// TIA Portal project "motor test code" (V20)

(* hardware
DEVICE "S7-1200 station_1"  S7-1200 Station
   slot 0: "Rack_0"  S7-1200 Rack  Rack  V1.0
   slot 1: "PLC_1"  CPU 1214C DC/DC/DC  6ES7 214-1AG40-0XB0  V4.6
   slot 2: "DI 8x24VDC/DQ 8xRelay_1"  SM 1223 DI8/DQ8 x relay  6ES7 223-1PH32-0XB0  V2.0
   slot 3: "AI 4x13BIT/AQ 2x14BIT_1"  SM 1234 AI4/AQ2  6ES7 234-4HE32-0XB0  V2.1
DEVICE "HMI_1"  KTP700 Basic PN
   slot 0: "HMI_1"  KTP700 Basic PN  6AV2 123-2GB03-0AX0  17.0.0.0
   slot 1: "HMI_RT_1"  KTP700 Basic PN  6AV2 123-2GB03-0AX0  17.0.0.0
   slot 5: "HMI_1.IE_CP_1"  PROFINET Interface  17.0.0.0
      slot 1: "PROFINET Interface_1"  PROFINET Interface
         slot 1: "Port_1"  Port
DEVICE "SINAMICS S_2"  SINAMICS S210
   slot 0: "Drive unit_2"  S210 PN  6SL3210-5HB10-4xFx  V5.2
      slot 1: "PROFINET interface"  PROFINET
      slot 3: "Ethernet commissioning interface"  LAN
   slot 0: "Drive control"  S210 PN
      slot 200: "Power Module_1"  Drive control  6SL3210-5HB10-4xFx
      slot 300: "Encoder evaluation_1"  Drive control  1FK2103-4AG0x-xMxx
      slot 400: "Measuring system_1"  Drive control  1FK2103-4AG0x-xMxx
      slot 1000: "Motor_1"  Drive control  1FK2103-4AG0x-xMxx
*)

// ===== PLC "PLC_1"  CPU 1214C DC/DC/DC =====

VAR_GLOBAL   // PLC tag table "Default tag table"
   "Brugaansturing_axis_IN" AT %I256.0 : "PD_TEL3_IN";
   "Brugaansturing_axis_OUT" AT %Q256.0 : "PD_TEL3_OUT";
   "ProgramCounter" AT %MW100 : Int;
   "em_stop" AT %I0.0 : Bool;
   "Reset Button" AT %I0.1 : Bool;
   "Homing sensor" AT %I0.2 : Bool;
   "Gate Closed" AT %I0.3 : Bool;
   "Gate Open" AT %I0.4 : Bool;
   "LightSwitch Front" AT %I0.5 : Bool;
   "LightSwitch Middle" AT %I0.6 : Bool;
   "Start Button" AT %I0.7 : Bool;
   "Stop Button" AT %I1.0 : Bool;
   "Open Gate" AT %Q0.0 : Bool;
   "Road_Yellow" AT %Q0.1 : Bool;
   "Road_Green" AT %Q0.2 : Bool;
   "Road_Red" AT %Q0.3 : Bool;
   "Noodstop Rood" AT %Q0.4 : Bool;
   "Noodstop Groen" AT %Q0.5 : Bool;
   "Autohome" AT %M1.1 : Bool;
   "JogForward" AT %M1.2 : Bool;
   "JogBackward" AT %M1.3 : Bool;
END_VAR

DATA_BLOCK "BrugAansturing_axis"   // DB1, Motion_DB
{ S7_Optimized_Access := 'TRUE' }
AUTHOR : SIMATIC
FAMILY : BasicMC
NAME : TO_PosAx
VERSION : 6.0
// stored: InstanceOfName TO_PositioningAxis
"TO_PositioningAxis"
BEGIN
   // Axis.Encoder.TelegramAddressOutCU = %Q256.0
   // Axis.Encoder.TelegramAddressInCU = %I256.0
   // Axis.Encoder.DoNameCU = Drive unit_2.Drive_control_Standard_telegram_3
   // Axis.Drive.TelegramAddressOutCU = %Q256.0
   // Axis.Drive.TelegramAddressInCU = %I256.0
   // Axis.Drive.TelegramType = 2
   // Axis.Drive.DoNameCU = Drive unit_2.Drive_control_Standard_telegram_3
   // Axis.Encoder.SelectedHscIndexCU = -1
   // Axis.LengthUnit.LastDistance = 1005
   // Axis.LengthUnitNormalized.Time = 1
   // Axis.LengthUnitNormalized.Distance = -2
   // Axis.Encoder.DbTypeCU = Classic
   // Axis.Drive.DbTypeCU = Classic
END_DATA_BLOCK

FUNCTION "Block_1" : Void   // FC1, SCL
{ S7_Optimized_Access := 'TRUE' }
VERSION : 0.1
BEGIN
   "MC_Home_DB"(Axis:="BrugAansturing_axis",
                Execute:="Autohome",
                Mode:=3);
   IF "BrugAansturing_axis".StatusBits.HomingDone THEN
       "Autohome" := 0
       ;
   END_IF;
END_FUNCTION

FUNCTION "my_function1" : Void   // FC2, SCL
{ S7_Optimized_Access := 'TRUE' }
VERSION : 0.1
BEGIN
   IF "JogForward"=TRUE THEN
       "MC_Halt_DB"(Axis := "BrugAansturing_axis",
                    Execute := FALSE);
       "MC_MoveVelocity_DB"(Axis := "BrugAansturing_axis",
                            Execute := TRUE,
                            Velocity := 40,
                            Direction := 0);

   ELSIF "JogBackward"=TRUE THEN
       "MC_Halt_DB"(Axis := "BrugAansturing_axis",
                    Execute := FALSE);
       "MC_MoveVelocity_DB"(Axis:="BrugAansturing_axis",
                              Execute:=TRUE,
                              Velocity:=-40,
                              Direction:=0);
     ELSE
         ;
         "MC_MoveVelocity_DB"(Axis := "BrugAansturing_axis",
                              Execute := FALSE);
         "MC_Halt_DB"(Axis:="BrugAansturing_axis",
                      Execute:=TRUE);

   END_IF;
END_FUNCTION

ORGANIZATION_BLOCK "Main"   // OB1, LAD, ProgramCycle
TITLE = "Main Program Sweep (Cycle)"
{ S7_Optimized_Access := 'TRUE' }
VERSION : 0.1
   VAR_INPUT
      Initial_Call : Bool;   // Initial call of this OB
      Remanence : Bool;   // =True, if remanent data are available
   END_VAR
BEGIN

REGION Network 1
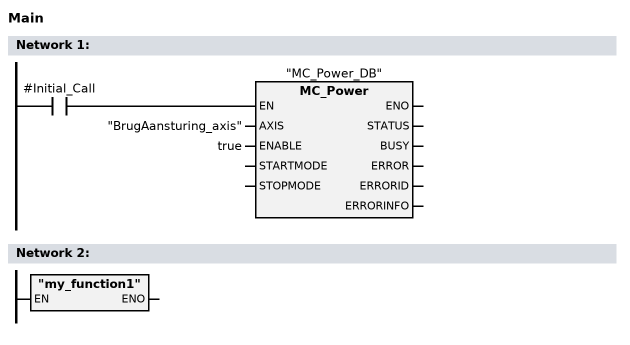
   IF #Initial_Call THEN
       "MC_Power_DB"(Axis := "BrugAansturing_axis", Enable := true);   // MC_Power
   END_IF;
END_REGION

REGION Network 2
   RUNG wire#powerrail
      "my_function1"()
   END_RUNG
   // the same network as SCL:
   "my_function1"();
END_REGION
END_ORGANIZATION_BLOCK

(* ===== HMI "HMI_RT_1" =====
system functions are stored by id; their names below are inferred from use
connection "HMI_Connection_1": ETHERNET, SMART_S7_1200_OMS

HMI tags "Default tag table"
   "HMI_Home" : UInt, internal
   "HMI_Debug" : UInt, internal
   "HMI_Manual overide" : UInt, internal
   "HMI_Nominal mode" : UInt, internal
   "em_stop" : Bool = PLC em_stop AT %I0.0, 100 ms
   "Homing sensor" : Bool = PLC "Homing sensor" AT %I0.2, 100 ms
   "Gate Closed" : Bool = PLC "Gate Closed" AT %I0.3, 100 ms
   "Gate Open" : Bool = PLC "Gate Open" AT %I0.4, 100 ms
   "ProgramCounter" : Int = PLC ProgramCounter AT %MW100, 100 ms
   "Autohome" : Bool = PLC Autohome AT %M1.1, 1 s
   "JogForward" : Bool = PLC JogForward AT %M1.2, 100 ms
   "JogBackward" : Bool = PLC JogBackward AT %M1.3, 100 ms

Template "Template_1" 800x480
   Button "Exit" at 714,429 size 71x50; TextOff 'Exit'; PictureOff "ExitRuntime_KTP700_Basic_PN_TR"; PictureOn "ExitRuntime_KTP700_Basic_PN_TR"
      on Release: StopRuntime(0)
   Button "Template_Button" at 614,429 size 71x50; TextOff 'Text'
   Button "Template_Button_1" at 514,429 size 71x50; TextOff 'Text'
   Button "Template_Button_2" at 414,429 size 71x50; TextOff 'Text'
   Button "Template_Button_3" at 314,429 size 71x50; TextOff 'Text'
   Button "Template_Button_4" at 214,429 size 71x50; TextOff 'Text'
   Button "Alarms" at 114,429 size 71x50; TextOff 'Alarms'; PictureOff "AlarmDisplay_KTP700_Basic_PN_TR"; PictureOn "AlarmDisplay_KTP700_Basic_PN_TR"
      on Release: function_ef3f5d25("Alarm window_Unacknowledged", -1)
   SymbolicIOField "Symbolic_IO_Field_Screen" at 93,9 size 600x33; TextOff '0'; TextOn '1'; TextList "TextList_ScreenNames"
      ProcessValue <- "HMI_Home"
      on Change: ActivateScreenByNumber("HMI_Home", 0)
   DateTimeField "HmiScreenItemData" at 695,25 size 105x25
   DateTimeField "HmiScreenItemData_1" at 695,0 size 105x25
   GraphicView "Logo" at 0,0 size 91x51; Picture "Logo of HMI_1"

screen "Home" 800x480, template "Template_1"
   on GenerateScreen: SetTag("HMI_Home", 2)
   TextField "HmiScreenItemData" at 71,58 size 640x43; Text 'Home'
   Button "Button_1" at 312,240 size 158x32; TextOff 'Debug'
      on Release: ActivateScreen("Debug", 0)
   TextField "Text field_1" at 312,192 size 152x23; Text 'Select your mode:'
   Button "Button_2" at 312,288 size 160x32; TextOff 'Manual Overide'
      on Release: ActivateScreen("Manual Overide", 0)
   Button "Button_3" at 312,336 size 160x32; TextOff 'Nominal Mode'
      on Release: ActivateScreen("Nominal Mode", 0)
   Button "Button_4" at 624,360 size 120x40; TextOff 'AutoHome'
      on Release: SetBit("Autohome")
   GraphicView "Graphic view_1" at 752,224 size 26x22; Picture "Graphic_1"
   GraphicView "Graphic view_2" at 736,192 size 35x35; Picture "Graphic_2"
   GraphicView "Graphic view_3" at 736,160 size 56x40; Picture "Graphic_3"
   GraphicView "Graphic view_4" at 720,176 size 44x32; Picture "Graphic_4"
   GraphicView "Graphic view_5" at 600,136 size 100x100; Picture "Graphic_5"
   TextField "Text field_2" at 536,224 size 221x23; Text 'Are you sure to AutoHome'
   Button "Button_5" at 664,280 size 96x32; TextOff 'NO'
   Button "Button_6" at 536,280 size 96x32; TextOff 'YES'

screen "Debug" 800x480, template "Template_1"
   on GenerateScreen: SetTag("HMI_Home", 3)
   TextField "HmiScreenItemData" at 77,51 size 640x51; Text 'Debug'
   Button "Back" at 1,52 size 159x47; TextOff 'Back'
      on Release: ActivateScreen("Home", 0)
   Circle "Circle_1" at 160,147 size 48x48
      Appearance <- "em_stop"
   Circle "Circle_2" at 157,215 size 48x48
      Appearance <- "Homing sensor"
   TextField "Text field_1" at 77,171 size 82x23; Text 'Noodstop'
   TextField "Text field_2" at 29,239 size 127x23; Text 'Homing Sensor'
   Circle "Circle_3" at 157,283 size 48x48
      Appearance <- "Gate Open"
   Circle "Circle_4" at 156,355 size 48x48
      Appearance <- "Gate Closed"
   TextField "Text field_3" at 26,307 size 130x23; Text 'Slagboom open'
   TextField "Text field_4" at 26,380 size 130x23; Text 'Slagboom dicht'
   IOField "I/O field_1" at 589,206 size 96x32; FormatPattern s999
      ProcessValue <- "ProgramCounter"
      Appearance <- "ProgramCounter"
   TextField "Text field_5" at 435,210 size 145x23; Text 'Program Counter'

screen "Nominal Mode" 800x480, template "Template_1"
   on GenerateScreen: SetTag("HMI_Home", 4)
   TextField "HmiScreenItemData" at 59,41 size 640x68; Text 'Nominal Mode'
   Button "Back" at 1,52 size 159x47; TextOff 'Back'
      on Release: ActivateScreen("Debug", 0)

screen "Manual Overide" 800x480, template "Template_1"
   on GenerateScreen: SetTag("HMI_Home", 5)
   TextField "HmiScreenItemData" at 81,35 size 640x49; Text 'Manual overide'
   Button "Back" at 1,52 size 159x47; TextOff 'Back'
      on Release: ActivateScreen("Nominal Mode", 0)
   Button "Button_2" at 296,232 size 200x56; TextOff 'JogBackward'
      on Press: function_b14e0dd5("JogBackward", 0)
      on Release: ResetBit("JogBackward")
   Button "Button_3" at 296,160 size 200x56; TextOff 'JogForward'
      on Press: function_b14e0dd5("JogForward", 0)
      on Release: ResetBit("JogForward")
   Circle "Circle_1" at 520,168 size 48x48
      Appearance <- "JogForward"
   Circle "Circle_2" at 520,240 size 48x48
      Appearance <- "JogBackward"
*)